PROGRAM MAIN
VAR
	Machine : FB_Machine;
	ControlSource : FB_ControlSource;
END_VAR

IF _TaskInfo[1].FirstCycle THEN
	Machine.RegisterExternalController(ControlSource);
END_IF


Machine.CyclicLogic();
ControlSource.CyclicLogic();

END_PROGRAM

(* stored: Version 1.1.0.1, ProductVersion 3.1.4024.12
   POU MAIN: Id {a42bdb35-f349-4c08-b658-08641a64a249}, SpecialFunc None *)
